// TIA Portal project "P2" (V20)

(* hardware
DEVICE "S7-1200 station_1"  S7-1200 Station
   slot 0: "Rack_0"  S7-1200 Rack  Rack  V1.0
   slot 1: "PLC_1"  CPU 1211C DC/DC/DC  6ES7 211-1AE40-0XB0  V4.7
*)

// ===== PLC "PLC_1"  CPU 1211C DC/DC/DC =====

VAR_GLOBAL   // PLC tag table "Default tag table"
   "Tag_1" AT %I0.0 : Bool;
   "Tag_2" AT %M0.1 : Bool;
   "Tag_3" AT %M0.0 : Bool;
   "Tag_4" AT %Q0.0 : Bool;
   "Tag_5" AT %Q0.1 : Bool;
END_VAR

ORGANIZATION_BLOCK "Main"   // OB1, LAD, ProgramCycle
TITLE = "Main Program Sweep (Cycle)"
{ S7_Optimized_Access := 'TRUE' }
VERSION : 0.1
   VAR_INPUT
      Initial_Call : Bool;   // Initial call of this OB
      Remanence : Bool;   // =True, if remanent data are available
   END_VAR
BEGIN

REGION Network 1
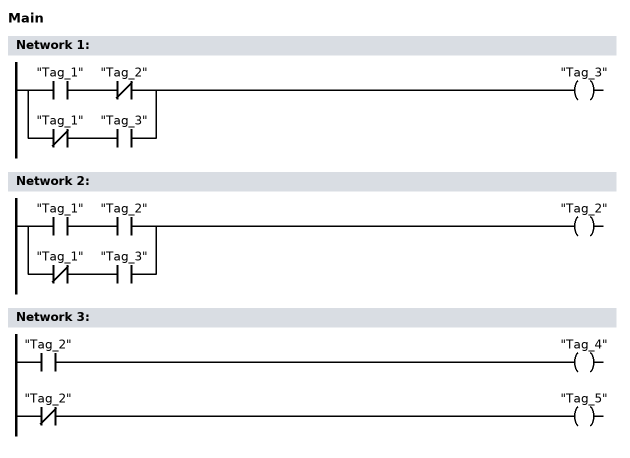
   RUNG wire#powerrail
      Contact( "Tag_1" )
      I_Contact( "Tag_2" )
      wire#w1
      Coil( "Tag_3" )
   END_RUNG
   RUNG wire#powerrail
      I_Contact( "Tag_1" )
      Contact( "Tag_3" )
   END_RUNG wire#w1
   // the same network as SCL:
   "Tag_3" := ("Tag_1" AND NOT "Tag_2") OR (NOT "Tag_1" AND "Tag_3");
END_REGION

REGION Network 2
   RUNG wire#powerrail
      Contact( "Tag_1" )
      Contact( "Tag_2" )
      wire#w1
      Coil( "Tag_2" )
   END_RUNG
   RUNG wire#powerrail
      I_Contact( "Tag_1" )
      Contact( "Tag_3" )
   END_RUNG wire#w1
   // the same network as SCL:
   "Tag_2" := ("Tag_1" AND "Tag_2") OR (NOT "Tag_1" AND "Tag_3");
END_REGION

REGION Network 3
   RUNG wire#powerrail
      Contact( "Tag_2" )
      Coil( "Tag_4" )
   END_RUNG
   RUNG wire#powerrail
      I_Contact( "Tag_2" )
      Coil( "Tag_5" )
   END_RUNG
   // the same network as SCL:
   "Tag_4" := "Tag_2";
   "Tag_5" := NOT "Tag_2";
END_REGION
END_ORGANIZATION_BLOCK